{attribute 'GeneratedUsingTerminal: EK1122-0000-0018'}
{attribute addProperty BoxType "EK1122-0000-0018"}
{attribute addProperty Id "Beckhoff_EL73xxsub_EK1100EK1100_1FC0878B2"}
{attribute addProperty CRC "3545871337"}
{attribute addProperty Size "2"}
{attribute addProperty Name "Beckhoff EL73xxEK1122"}
TYPE Beckhoff_EL73xxEK1122_D359B3E9 EXTENDS EK1122_1FC0878B :
STRUCT
	{attribute addProperty Name "Beckhoff EL73xxsub EK1100"}
	{attribute addProperty PreviousPort "Beckhoff EL73xxEK1122 : D"}
	Beckhoff_EL73xxsub_EK1100 : EK1100_1FC0878B;
END_STRUCT
END_TYPE

(* stored: Version 1.2.0.0, ProductVersion 3.1.4024.11
   DUT Beckhoff_EL73xxEK1122_D359B3E9: Id {0ac5a338-f724-425d-9799-da4c513118ea} *)
